{attribute 'qualified_only'}
{attribute 'strict'}
TYPE ENUM_SolidAttenuator_Staes :
(

    Unknown := 0,
    OUT := 1,
    Target1 := 2,
    Target2 := 3,
    Target3 := 4,
    Target4 := 5,
    Target5 := 6

)UINT;
END_TYPE

(* stored: Version 1.1.0.1, ProductVersion 3.1.4022.18
   DUT ENUM_SolidAttenuator_Staes: Id {a9b56f49-37af-4519-bf3c-f4ee10056eb1} *)
